INTERFACE ITF_BaseGroupElementDecoratorParent EXTENDS ITF_BaseGroupElement

END_INTERFACE

(* stored: Version 1.1.0.1
   Itf ITF_BaseGroupElementDecoratorParent: Id {a829f283-48ff-04f8-26c1-bceded6302ed} *)
